TYPE ST_M001_IO_OUT :
STRUCT
END_STRUCT
END_TYPE

(* stored: Version 1.1.0.1
   DUT ST_M001_IO_OUT: Id {dbf409dd-0212-4396-a59e-0978c91af846} *)
